% RSLogix 500 project Adaptive Fault-Resilient Robotic Pick-and-Place Cell.RSS, saved by version 8.30.00.16 %
PROJECT "UNTITLED"    % processor: Bul.1763 MicroLogix 1100 Series B %

PROGRAM FILES
  LAD 2 "MAIN/ARM"  15 rungs
  LAD 3 "SAFETY"  28 rungs
  LAD 4 "MODES"  4 rungs
  LAD 5 "DIGITAL IO"  17 rungs
  LAD 6 "ANALOG IO"  2 rungs
  LAD 7 "STATE"  6 rungs
  LAD 8 "SENSORS"  5 rungs
  LAD 9 "SYSTEM H"  6 rungs
  LAD 10 "H SAFETY"  6 rungs
  LAD 11 "H IO"  3 rungs
  LAD 12 "H STATE"  4 rungs
  LAD 13 "LOGIC"  19 rungs

DATA FILES
  O0 OUTPUT  7 elements
  I1 INPUT  14 elements
  S2 STATUS  66 elements
  B3 BINARY  10 elements
  T4 TIMER  8 elements
  C5 COUNTER  10 elements
  R6 CONTROL  1 elements
  N7 INTEGER  1 elements
  F8 FLOAT  1 elements

LADDER 2 "MAIN/ARM"
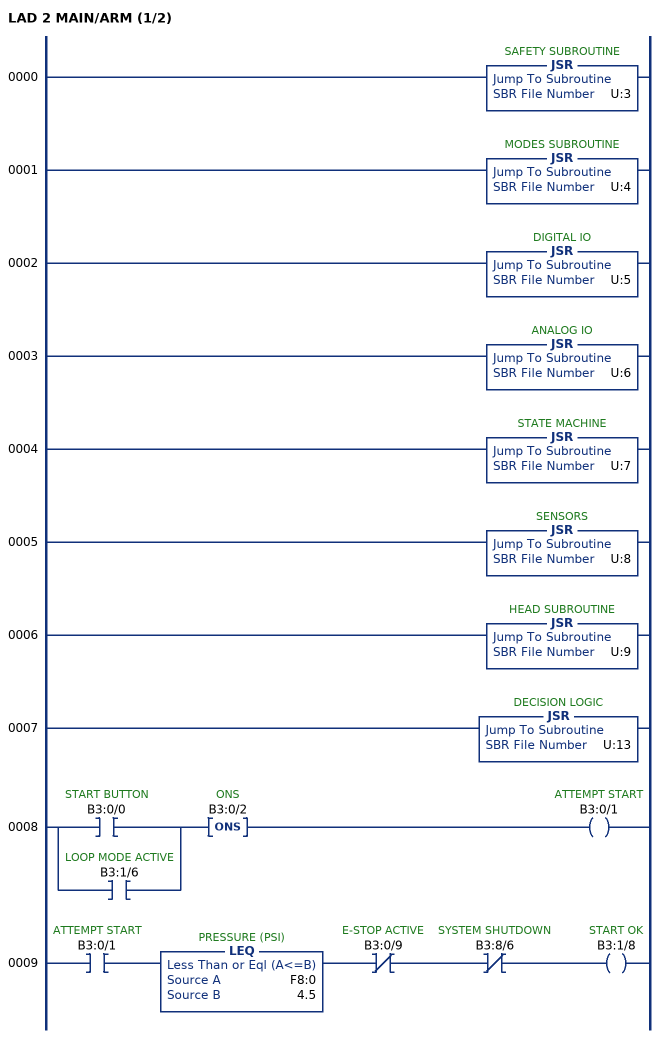
% Rung: 0 %
SOR JSR U:3 EOR
%   U:3  "SAFETY SUBROUTINE" %
% Rung: 1 %
SOR JSR U:4 EOR
%   U:4  "MODES SUBROUTINE" %
% Rung: 2 %
SOR JSR U:5 EOR
%   U:5  "DIGITAL IO" %
% Rung: 3 %
SOR JSR U:6 EOR
%   U:6  "ANALOG IO" %
% Rung: 4 %
SOR JSR U:7 EOR
%   U:7  "STATE MACHINE" %
% Rung: 5 %
SOR JSR U:8 EOR
%   U:8  "SENSORS" %
% Rung: 6 %
SOR JSR U:9 EOR
%   U:9  "HEAD SUBROUTINE" %
% Rung: 7 %
SOR JSR U:13 EOR
%   U:13  "DECISION LOGIC" %
% Rung: 8 %
SOR BST XIC B3:0/0 NXB XIC B3:1/6 BND ONS B3:0/2 OTE B3:0/1 EOR
%   B3:0/0  "START BUTTON" %
%   B3:1/6  "LOOP MODE ACTIVE" %
%   B3:0/2  "ONS" %
%   B3:0/1  "ATTEMPT START" %
% Rung: 9 %
SOR XIC B3:0/1 LEQ F8:0 4.5 XIO B3:0/9 XIO B3:8/6 OTE B3:1/8 EOR
%   B3:0/1  "ATTEMPT START" %
%   F8:0  "PRESSURE (PSI)" %
%   B3:0/9  "E-STOP ACTIVE" %
%   B3:8/6  "SYSTEM SHUTDOWN" %
%   B3:1/8  "START OK" %

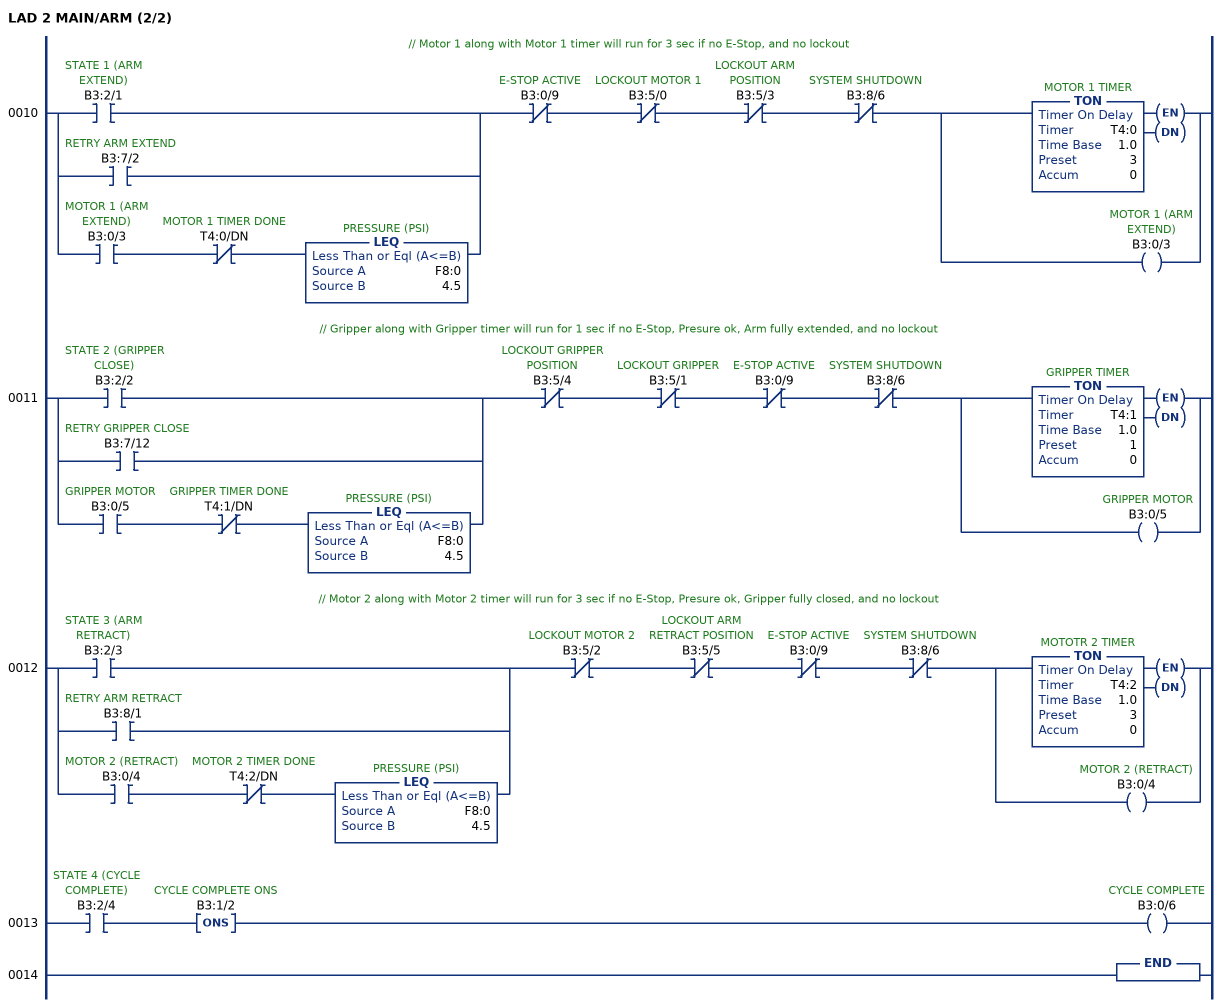
% Rung: 10 %
% // Motor 1 along with Motor 1 timer will run for 3 sec if no E-Stop, and no lockout %
SOR BST BST XIC B3:2/1 NXB XIC B3:7/2 BND NXB XIC B3:0/3 XIO T4:0/DN LEQ F8:0 4.5 BND XIO B3:0/9 XIO B3:5/0 XIO B3:5/3 XIO B3:8/6 BST TON T4:0 1.0 3 0 NXB OTE B3:0/3 BND EOR
%   B3:2/1  "STATE 1 (ARM EXTEND)" %
%   B3:7/2  "RETRY ARM EXTEND" %
%   B3:0/3  "MOTOR 1 (ARM EXTEND)" %
%   T4:0/DN  "MOTOR 1 TIMER DONE" %
%   F8:0  "PRESSURE (PSI)" %
%   B3:0/9  "E-STOP ACTIVE" %
%   B3:5/0  "LOCKOUT MOTOR 1" %
%   B3:5/3  "LOCKOUT ARM POSITION" %
%   B3:8/6  "SYSTEM SHUTDOWN" %
%   T4:0  "MOTOR 1 TIMER" %
% Rung: 11 %
% // Gripper along with Gripper timer will run for 1 sec if no E-Stop, Presure ok, Arm fully extended, and no lockout %
SOR BST BST XIC B3:2/2 NXB XIC B3:7/12 BND NXB XIC B3:0/5 XIO T4:1/DN LEQ F8:0 4.5 BND XIO B3:5/4 XIO B3:5/1 XIO B3:0/9 XIO B3:8/6 BST TON T4:1 1.0 1 0 NXB OTE B3:0/5 BND EOR
%   B3:2/2  "STATE 2 (GRIPPER CLOSE)" %
%   B3:7/12  "RETRY GRIPPER CLOSE" %
%   B3:0/5  "GRIPPER MOTOR" %
%   T4:1/DN  "GRIPPER TIMER DONE" %
%   F8:0  "PRESSURE (PSI)" %
%   B3:5/4  "LOCKOUT GRIPPER POSITION" %
%   B3:5/1  "LOCKOUT GRIPPER" %
%   B3:0/9  "E-STOP ACTIVE" %
%   B3:8/6  "SYSTEM SHUTDOWN" %
%   T4:1  "GRIPPER TIMER" %
% Rung: 12 %
% // Motor 2 along with Motor 2 timer will run for 3 sec if no E-Stop, Presure ok, Gripper fully closed, and no lockout %
SOR BST BST XIC B3:2/3 NXB XIC B3:8/1 BND NXB XIC B3:0/4 XIO T4:2/DN LEQ F8:0 4.5 BND XIO B3:5/2 XIO B3:5/5 XIO B3:0/9 XIO B3:8/6 BST TON T4:2 1.0 3 0 NXB OTE B3:0/4 BND EOR
%   B3:2/3  "STATE 3 (ARM RETRACT)" %
%   B3:8/1  "RETRY ARM RETRACT" %
%   B3:0/4  "MOTOR 2 (RETRACT)" %
%   T4:2/DN  "MOTOR 2 TIMER DONE" %
%   F8:0  "PRESSURE (PSI)" %
%   B3:5/2  "LOCKOUT MOTOR 2" %
%   B3:5/5  "LOCKOUT ARM RETRACT POSITION" %
%   B3:0/9  "E-STOP ACTIVE" %
%   B3:8/6  "SYSTEM SHUTDOWN" %
%   T4:2  "MOTOTR 2 TIMER" %
% Rung: 13 %
SOR XIC B3:2/4 ONS B3:1/2 OTE B3:0/6 EOR
%   B3:2/4  "STATE 4 (CYCLE COMPLETE)" %
%   B3:1/2  "CYCLE COMPLETE ONS" %
%   B3:0/6  "CYCLE COMPLETE" %
% Rung: 14 %
SOR END EOR

LADDER 3 "SAFETY"
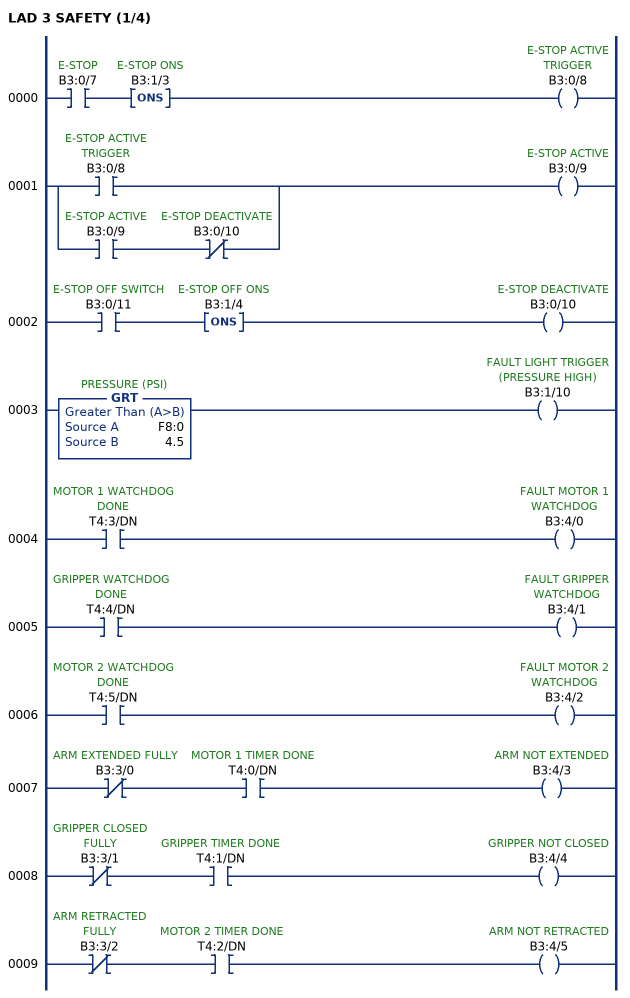
% Rung: 0 %
SOR XIC B3:0/7 ONS B3:1/3 OTE B3:0/8 EOR
%   B3:0/7  "E-STOP" %
%   B3:1/3  "E-STOP ONS" %
%   B3:0/8  "E-STOP ACTIVE TRIGGER" %
% Rung: 1 %
SOR BST XIC B3:0/8 NXB XIC B3:0/9 XIO B3:0/10 BND OTE B3:0/9 EOR
%   B3:0/8  "E-STOP ACTIVE TRIGGER" %
%   B3:0/9  "E-STOP ACTIVE" %
%   B3:0/10  "E-STOP DEACTIVATE" %
% Rung: 2 %
SOR XIC B3:0/11 ONS B3:1/4 OTE B3:0/10 EOR
%   B3:0/11  "E-STOP OFF SWITCH" %
%   B3:1/4  "E-STOP OFF ONS" %
%   B3:0/10  "E-STOP DEACTIVATE" %
% Rung: 3 %
SOR GRT F8:0 4.5 OTE B3:1/10 EOR
%   F8:0  "PRESSURE (PSI)" %
%   B3:1/10  "FAULT LIGHT TRIGGER (PRESSURE HIGH)" %
% Rung: 4 %
SOR XIC T4:3/DN OTE B3:4/0 EOR
%   T4:3/DN  "MOTOR 1 WATCHDOG DONE" %
%   B3:4/0  "FAULT MOTOR 1 WATCHDOG" %
% Rung: 5 %
SOR XIC T4:4/DN OTE B3:4/1 EOR
%   T4:4/DN  "GRIPPER WATCHDOG DONE" %
%   B3:4/1  "FAULT GRIPPER WATCHDOG" %
% Rung: 6 %
SOR XIC T4:5/DN OTE B3:4/2 EOR
%   T4:5/DN  "MOTOR 2 WATCHDOG DONE" %
%   B3:4/2  "FAULT MOTOR 2 WATCHDOG" %
% Rung: 7 %
SOR XIO B3:3/0 XIC T4:0/DN OTE B3:4/3 EOR
%   B3:3/0  "ARM EXTENDED FULLY" %
%   T4:0/DN  "MOTOR 1 TIMER DONE" %
%   B3:4/3  "ARM NOT EXTENDED" %
% Rung: 8 %
SOR XIO B3:3/1 XIC T4:1/DN OTE B3:4/4 EOR
%   B3:3/1  "GRIPPER CLOSED FULLY" %
%   T4:1/DN  "GRIPPER TIMER DONE" %
%   B3:4/4  "GRIPPER NOT CLOSED" %
% Rung: 9 %
SOR XIO B3:3/2 XIC T4:2/DN OTE B3:4/5 EOR
%   B3:3/2  "ARM RETRACTED FULLY" %
%   T4:2/DN  "MOTOR 2 TIMER DONE" %
%   B3:4/5  "ARM NOT RETRACTED" %

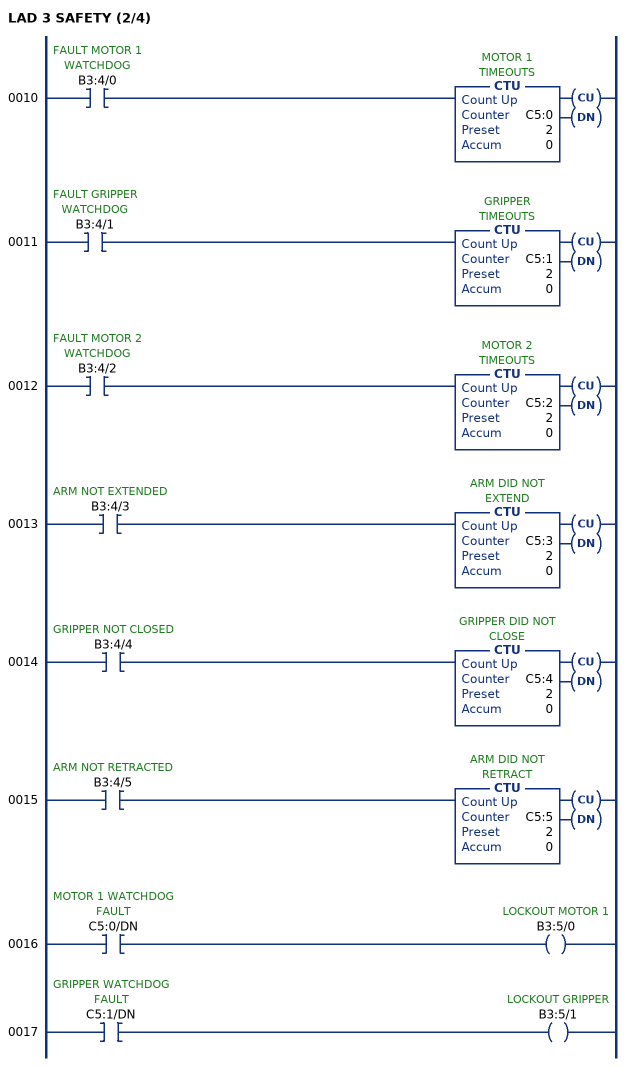
% Rung: 10 %
SOR XIC B3:4/0 CTU C5:0 2 0 EOR
%   B3:4/0  "FAULT MOTOR 1 WATCHDOG" %
%   C5:0  "MOTOR 1 TIMEOUTS" %
% Rung: 11 %
SOR XIC B3:4/1 CTU C5:1 2 0 EOR
%   B3:4/1  "FAULT GRIPPER WATCHDOG" %
%   C5:1  "GRIPPER TIMEOUTS" %
% Rung: 12 %
SOR XIC B3:4/2 CTU C5:2 2 0 EOR
%   B3:4/2  "FAULT MOTOR 2 WATCHDOG" %
%   C5:2  "MOTOR 2 TIMEOUTS" %
% Rung: 13 %
SOR XIC B3:4/3 CTU C5:3 2 0 EOR
%   B3:4/3  "ARM NOT EXTENDED" %
%   C5:3  "ARM DID NOT EXTEND" %
% Rung: 14 %
SOR XIC B3:4/4 CTU C5:4 2 0 EOR
%   B3:4/4  "GRIPPER NOT CLOSED" %
%   C5:4  "GRIPPER DID NOT CLOSE" %
% Rung: 15 %
SOR XIC B3:4/5 CTU C5:5 2 0 EOR
%   B3:4/5  "ARM NOT RETRACTED" %
%   C5:5  "ARM DID NOT RETRACT" %
% Rung: 16 %
SOR XIC C5:0/DN OTE B3:5/0 EOR
%   C5:0/DN  "MOTOR 1 WATCHDOG FAULT" %
%   B3:5/0  "LOCKOUT MOTOR 1" %
% Rung: 17 %
SOR XIC C5:1/DN OTE B3:5/1 EOR
%   C5:1/DN  "GRIPPER WATCHDOG FAULT" %
%   B3:5/1  "LOCKOUT GRIPPER" %

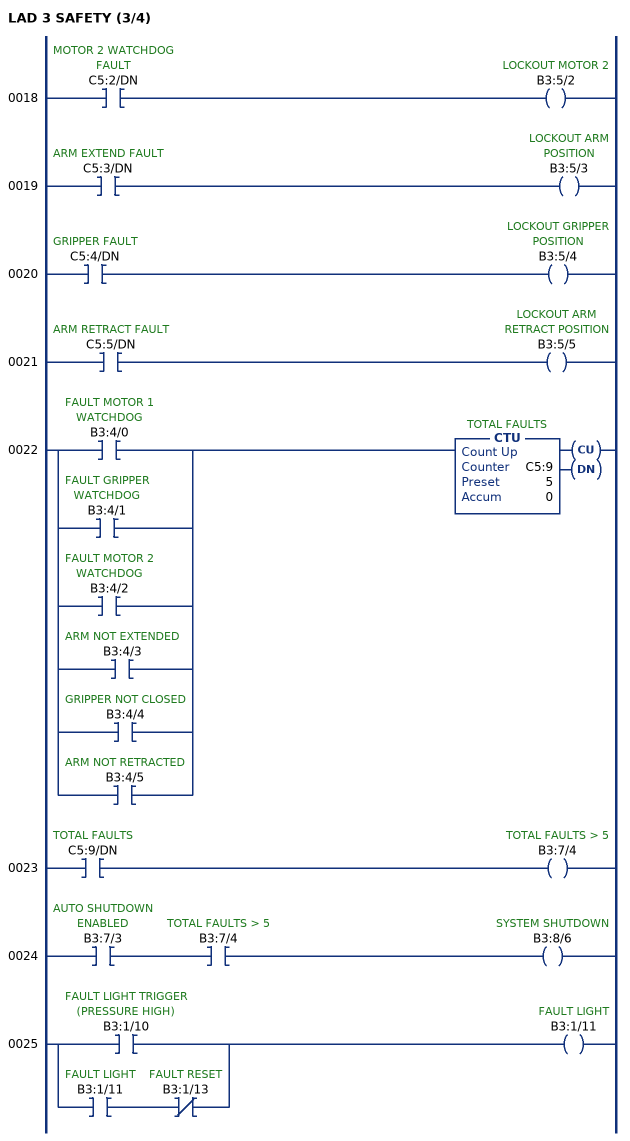
% Rung: 18 %
SOR XIC C5:2/DN OTE B3:5/2 EOR
%   C5:2/DN  "MOTOR 2 WATCHDOG FAULT" %
%   B3:5/2  "LOCKOUT MOTOR 2" %
% Rung: 19 %
SOR XIC C5:3/DN OTE B3:5/3 EOR
%   C5:3/DN  "ARM EXTEND FAULT" %
%   B3:5/3  "LOCKOUT ARM POSITION" %
% Rung: 20 %
SOR XIC C5:4/DN OTE B3:5/4 EOR
%   C5:4/DN  "GRIPPER FAULT" %
%   B3:5/4  "LOCKOUT GRIPPER POSITION" %
% Rung: 21 %
SOR XIC C5:5/DN OTE B3:5/5 EOR
%   C5:5/DN  "ARM RETRACT FAULT" %
%   B3:5/5  "LOCKOUT ARM RETRACT POSITION" %
% Rung: 22 %
SOR BST XIC B3:4/0 NXB XIC B3:4/1 NXB XIC B3:4/2 NXB XIC B3:4/3 NXB XIC B3:4/4 NXB XIC B3:4/5 BND CTU C5:9 5 0 EOR
%   B3:4/0  "FAULT MOTOR 1 WATCHDOG" %
%   B3:4/1  "FAULT GRIPPER WATCHDOG" %
%   B3:4/2  "FAULT MOTOR 2 WATCHDOG" %
%   B3:4/3  "ARM NOT EXTENDED" %
%   B3:4/4  "GRIPPER NOT CLOSED" %
%   B3:4/5  "ARM NOT RETRACTED" %
%   C5:9  "TOTAL FAULTS" %
% Rung: 23 %
SOR XIC C5:9/DN OTE B3:7/4 EOR
%   C5:9  "TOTAL FAULTS" %
%   B3:7/4  "TOTAL FAULTS > 5" %
% Rung: 24 %
SOR XIC B3:7/3 XIC B3:7/4 OTE B3:8/6 EOR
%   B3:7/3  "AUTO SHUTDOWN ENABLED" %
%   B3:7/4  "TOTAL FAULTS > 5" %
%   B3:8/6  "SYSTEM SHUTDOWN" %
% Rung: 25 %
SOR BST XIC B3:1/10 NXB XIC B3:1/11 XIO B3:1/13 BND OTE B3:1/11 EOR
%   B3:1/10  "FAULT LIGHT TRIGGER (PRESSURE HIGH)" %
%   B3:1/11  "FAULT LIGHT" %
%   B3:1/13  "FAULT RESET" %

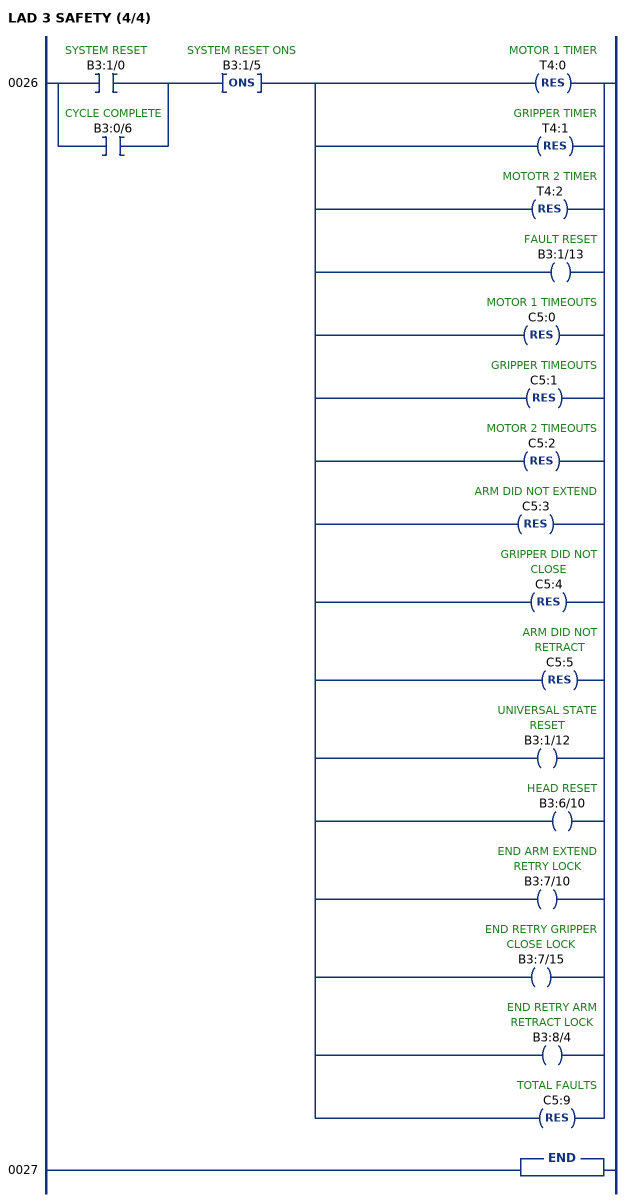
% Rung: 26 %
SOR BST XIC B3:1/0 NXB XIC B3:0/6 BND ONS B3:1/5 BST RES T4:0 NXB RES T4:1 NXB RES T4:2 NXB OTE B3:1/13 NXB RES C5:0 NXB RES C5:1 NXB RES C5:2 NXB RES C5:3 NXB RES C5:4 NXB RES C5:5 NXB OTE B3:1/12 NXB OTE B3:6/10 NXB OTE B3:7/10 NXB OTE B3:7/15 NXB OTE B3:8/4 NXB RES C5:9 BND EOR
%   B3:1/0  "SYSTEM RESET" %
%   B3:0/6  "CYCLE COMPLETE" %
%   B3:1/5  "SYSTEM RESET ONS" %
%   T4:0  "MOTOR 1 TIMER" %
%   T4:1  "GRIPPER TIMER" %
%   T4:2  "MOTOTR 2 TIMER" %
%   B3:1/13  "FAULT RESET" %
%   C5:0  "MOTOR 1 TIMEOUTS" %
%   C5:1  "GRIPPER TIMEOUTS" %
%   C5:2  "MOTOR 2 TIMEOUTS" %
%   C5:3  "ARM DID NOT EXTEND" %
%   C5:4  "GRIPPER DID NOT CLOSE" %
%   C5:5  "ARM DID NOT RETRACT" %
%   B3:1/12  "UNIVERSAL STATE RESET" %
%   B3:6/10  "HEAD RESET" %
%   B3:7/10  "END ARM EXTEND RETRY LOCK" %
%   B3:7/15  "END RETRY GRIPPER CLOSE LOCK" %
%   B3:8/4  "END RETRY ARM RETRACT LOCK" %
%   C5:9  "TOTAL FAULTS" %
% Rung: 27 %
SOR END EOR

LADDER 4 "MODES"
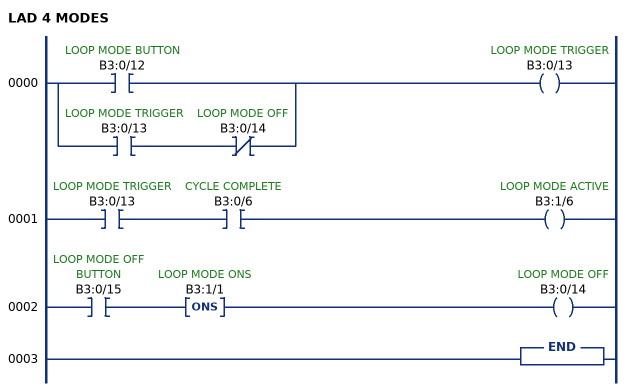
% Rung: 0 %
SOR BST XIC B3:0/12 NXB XIC B3:0/13 XIO B3:0/14 BND OTE B3:0/13 EOR
%   B3:0/12  "LOOP MODE BUTTON" %
%   B3:0/13  "LOOP MODE TRIGGER" %
%   B3:0/14  "LOOP MODE OFF" %
% Rung: 1 %
SOR XIC B3:0/13 XIC B3:0/6 OTE B3:1/6 EOR
%   B3:0/13  "LOOP MODE TRIGGER" %
%   B3:0/6  "CYCLE COMPLETE" %
%   B3:1/6  "LOOP MODE ACTIVE" %
% Rung: 2 %
SOR XIC B3:0/15 ONS B3:1/1 OTE B3:0/14 EOR
%   B3:0/15  "LOOP MODE OFF BUTTON" %
%   B3:1/1  "LOOP MODE ONS" %
%   B3:0/14  "LOOP MODE OFF" %
% Rung: 3 %
SOR END EOR

LADDER 5 "DIGITAL IO"
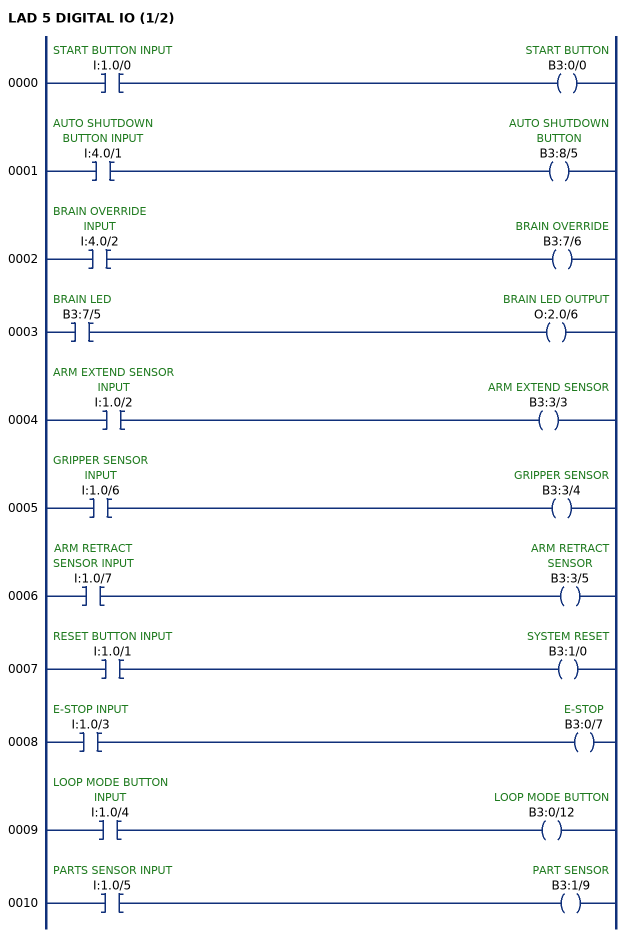
% Rung: 0 %
SOR XIC I:1.0/0 OTE B3:0/0 EOR
%   I:1.0/0  "START BUTTON INPUT" %
%   B3:0/0  "START BUTTON" %
% Rung: 1 %
SOR XIC I:4.0/1 OTE B3:8/5 EOR
%   I:4.0/1  "AUTO SHUTDOWN BUTTON INPUT" %
%   B3:8/5  "AUTO SHUTDOWN BUTTON" %
% Rung: 2 %
SOR XIC I:4.0/2 OTE B3:7/6 EOR
%   I:4.0/2  "BRAIN OVERRIDE INPUT" %
%   B3:7/6  "BRAIN OVERRIDE" %
% Rung: 3 %
SOR XIC B3:7/5 OTE O:2.0/6 EOR
%   B3:7/5  "BRAIN LED" %
%   O:2.0/6  "BRAIN LED OUTPUT" %
% Rung: 4 %
SOR XIC I:1.0/2 OTE B3:3/3 EOR
%   I:1.0/2  "ARM EXTEND SENSOR INPUT" %
%   B3:3/3  "ARM EXTEND SENSOR" %
% Rung: 5 %
SOR XIC I:1.0/6 OTE B3:3/4 EOR
%   I:1.0/6  "GRIPPER SENSOR INPUT" %
%   B3:3/4  "GRIPPER SENSOR" %
% Rung: 6 %
SOR XIC I:1.0/7 OTE B3:3/5 EOR
%   I:1.0/7  "ARM RETRACT SENSOR INPUT" %
%   B3:3/5  "ARM RETRACT SENSOR" %
% Rung: 7 %
SOR XIC I:1.0/1 OTE B3:1/0 EOR
%   I:1.0/1  "RESET BUTTON INPUT" %
%   B3:1/0  "SYSTEM RESET" %
% Rung: 8 %
SOR XIC I:1.0/3 OTE B3:0/7 EOR
%   I:1.0/3  "E-STOP INPUT" %
%   B3:0/7  "E-STOP" %
% Rung: 9 %
SOR XIC I:1.0/4 OTE B3:0/12 EOR
%   I:1.0/4  "LOOP MODE BUTTON INPUT" %
%   B3:0/12  "LOOP MODE BUTTON" %
% Rung: 10 %
SOR XIC I:1.0/5 OTE B3:1/9 EOR
%   I:1.0/5  "PARTS SENSOR INPUT" %
%   B3:1/9  "PART SENSOR" %

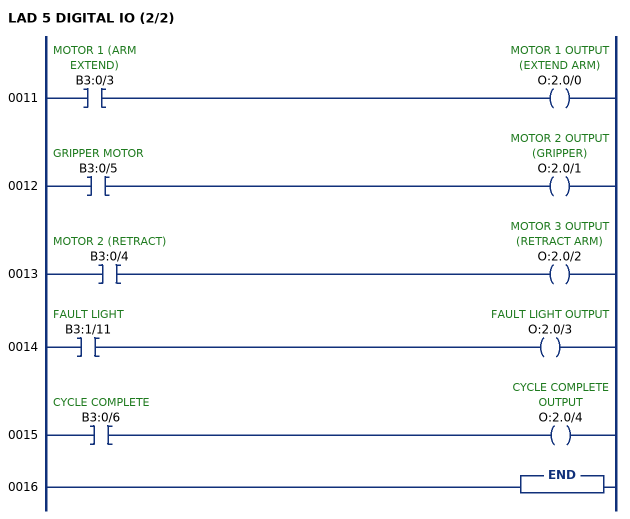
% Rung: 11 %
SOR XIC B3:0/3 OTE O:2.0/0 EOR
%   B3:0/3  "MOTOR 1 (ARM EXTEND)" %
%   O:2.0/0  "MOTOR 1 OUTPUT (EXTEND ARM)" %
% Rung: 12 %
SOR XIC B3:0/5 OTE O:2.0/1 EOR
%   B3:0/5  "GRIPPER MOTOR" %
%   O:2.0/1  "MOTOR 2 OUTPUT (GRIPPER)" %
% Rung: 13 %
SOR XIC B3:0/4 OTE O:2.0/2 EOR
%   B3:0/4  "MOTOR 2 (RETRACT)" %
%   O:2.0/2  "MOTOR 3 OUTPUT (RETRACT ARM)" %
% Rung: 14 %
SOR XIC B3:1/11 OTE O:2.0/3 EOR
%   B3:1/11  "FAULT LIGHT" %
%   O:2.0/3  "FAULT LIGHT OUTPUT" %
% Rung: 15 %
SOR XIC B3:0/6 OTE O:2.0/4 EOR
%   B3:0/6  "CYCLE COMPLETE" %
%   O:2.0/4  "CYCLE COMPLETE OUTPUT" %
% Rung: 16 %
SOR END EOR

LADDER 6 "ANALOG IO"
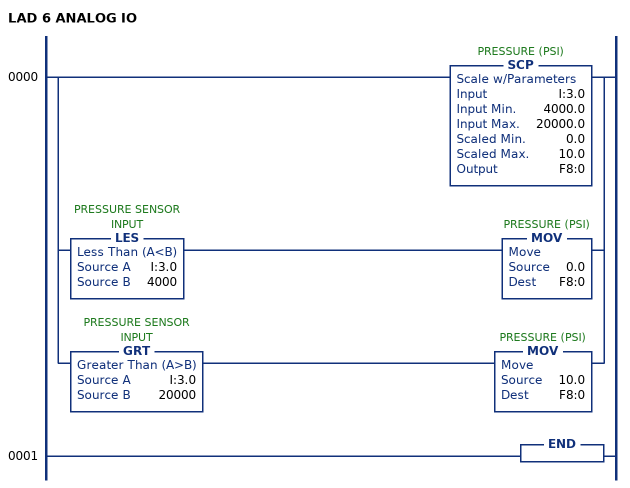
% Rung: 0 %
SOR BST SCP I:3.0 4000.0 20000.0 0.0 10.0 F8:0 NXB LES I:3.0 4000 MOV 0.0 F8:0 NXB GRT I:3.0 20000 MOV 10.0 F8:0 BND EOR
%   I:3.0  "PRESSURE SENSOR INPUT" %
%   F8:0  "PRESSURE (PSI)" %
% Rung: 1 %
SOR END EOR

LADDER 7 "STATE"
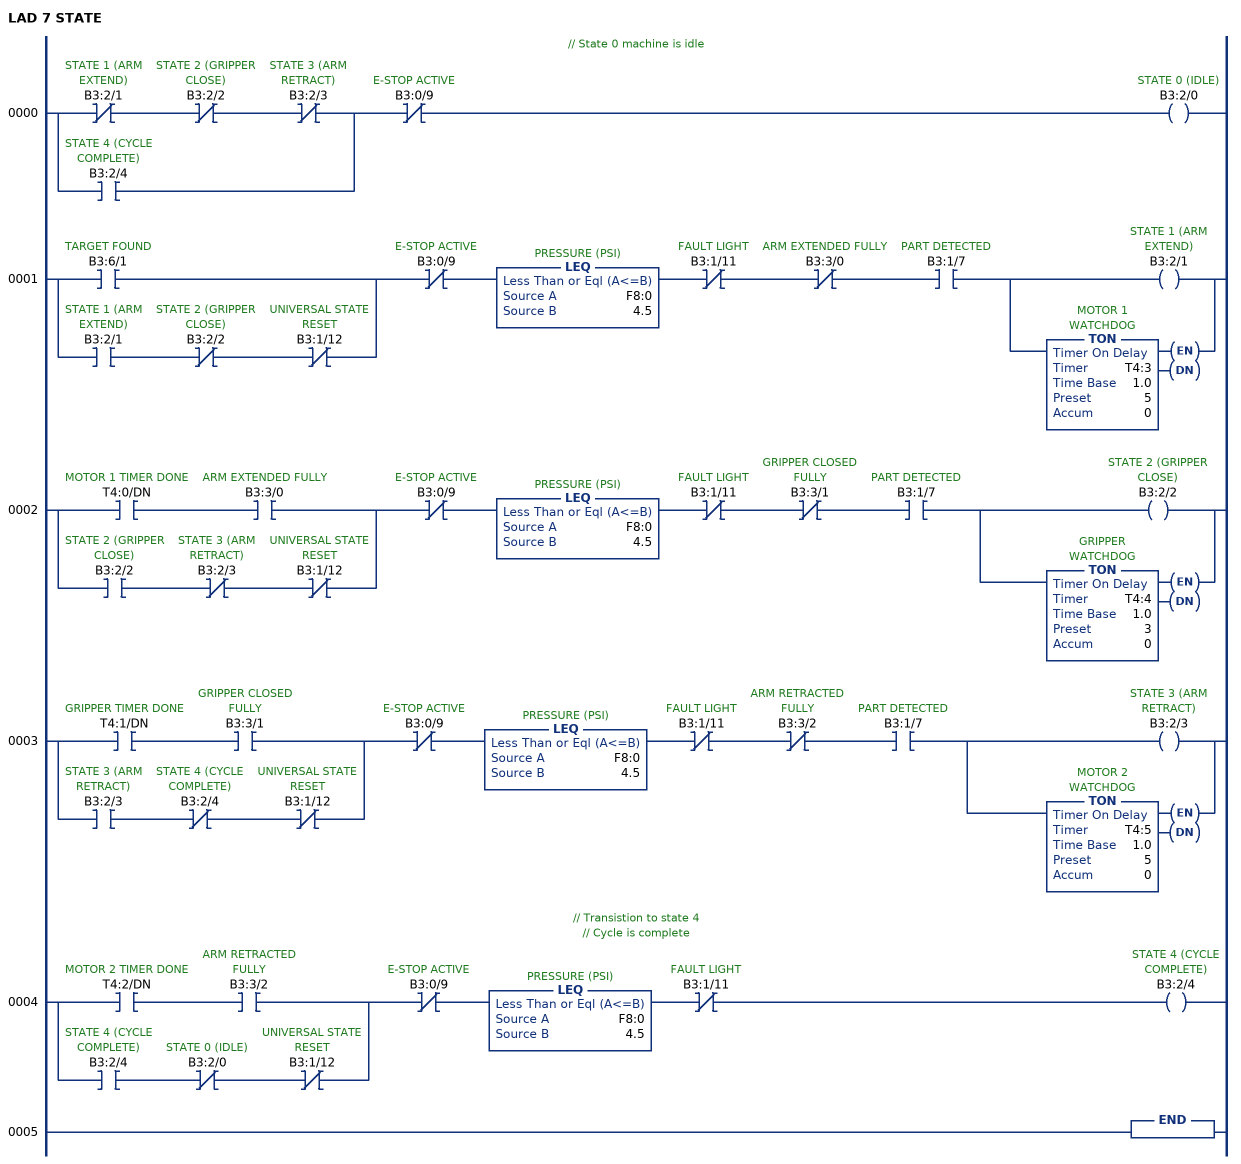
% Rung: 0 %
% // State 0 machine is idle %
SOR BST XIO B3:2/1 XIO B3:2/2 XIO B3:2/3 NXB XIC B3:2/4 BND XIO B3:0/9 OTE B3:2/0 EOR
%   B3:2/1  "STATE 1 (ARM EXTEND)" %
%   B3:2/2  "STATE 2 (GRIPPER CLOSE)" %
%   B3:2/3  "STATE 3 (ARM RETRACT)" %
%   B3:2/4  "STATE 4 (CYCLE COMPLETE)" %
%   B3:0/9  "E-STOP ACTIVE" %
%   B3:2/0  "STATE 0 (IDLE)" %
% Rung: 1 %
SOR BST XIC B3:6/1 NXB XIC B3:2/1 XIO B3:2/2 XIO B3:1/12 BND XIO B3:0/9 LEQ F8:0 4.5 XIO B3:1/11 XIO B3:3/0 XIC B3:1/7 BST OTE B3:2/1 NXB TON T4:3 1.0 5 0 BND EOR
%   B3:6/1  "TARGET FOUND" %
%   B3:2/1  "STATE 1 (ARM EXTEND)" %
%   B3:2/2  "STATE 2 (GRIPPER CLOSE)" %
%   B3:1/12  "UNIVERSAL STATE RESET" %
%   B3:0/9  "E-STOP ACTIVE" %
%   F8:0  "PRESSURE (PSI)" %
%   B3:1/11  "FAULT LIGHT" %
%   B3:3/0  "ARM EXTENDED FULLY" %
%   B3:1/7  "PART DETECTED" %
%   T4:3  "MOTOR 1 WATCHDOG" %
% Rung: 2 %
SOR BST XIC T4:0/DN XIC B3:3/0 NXB XIC B3:2/2 XIO B3:2/3 XIO B3:1/12 BND XIO B3:0/9 LEQ F8:0 4.5 XIO B3:1/11 XIO B3:3/1 XIC B3:1/7 BST OTE B3:2/2 NXB TON T4:4 1.0 3 0 BND EOR
%   T4:0/DN  "MOTOR 1 TIMER DONE" %
%   B3:3/0  "ARM EXTENDED FULLY" %
%   B3:2/2  "STATE 2 (GRIPPER CLOSE)" %
%   B3:2/3  "STATE 3 (ARM RETRACT)" %
%   B3:1/12  "UNIVERSAL STATE RESET" %
%   B3:0/9  "E-STOP ACTIVE" %
%   F8:0  "PRESSURE (PSI)" %
%   B3:1/11  "FAULT LIGHT" %
%   B3:3/1  "GRIPPER CLOSED FULLY" %
%   B3:1/7  "PART DETECTED" %
%   T4:4  "GRIPPER WATCHDOG" %
% Rung: 3 %
SOR BST XIC T4:1/DN XIC B3:3/1 NXB XIC B3:2/3 XIO B3:2/4 XIO B3:1/12 BND XIO B3:0/9 LEQ F8:0 4.5 XIO B3:1/11 XIO B3:3/2 XIC B3:1/7 BST OTE B3:2/3 NXB TON T4:5 1.0 5 0 BND EOR
%   T4:1/DN  "GRIPPER TIMER DONE" %
%   B3:3/1  "GRIPPER CLOSED FULLY" %
%   B3:2/3  "STATE 3 (ARM RETRACT)" %
%   B3:2/4  "STATE 4 (CYCLE COMPLETE)" %
%   B3:1/12  "UNIVERSAL STATE RESET" %
%   B3:0/9  "E-STOP ACTIVE" %
%   F8:0  "PRESSURE (PSI)" %
%   B3:1/11  "FAULT LIGHT" %
%   B3:3/2  "ARM RETRACTED FULLY" %
%   B3:1/7  "PART DETECTED" %
%   T4:5  "MOTOR 2 WATCHDOG" %
% Rung: 4 %
% // Transistion to state 4
% // Cycle is complete %
SOR BST XIC T4:2/DN XIC B3:3/2 NXB XIC B3:2/4 XIO B3:2/0 XIO B3:1/12 BND XIO B3:0/9 LEQ F8:0 4.5 XIO B3:1/11 OTE B3:2/4 EOR
%   T4:2/DN  "MOTOR 2 TIMER DONE" %
%   B3:3/2  "ARM RETRACTED FULLY" %
%   B3:2/4  "STATE 4 (CYCLE COMPLETE)" %
%   B3:2/0  "STATE 0 (IDLE)" %
%   B3:1/12  "UNIVERSAL STATE RESET" %
%   B3:0/9  "E-STOP ACTIVE" %
%   F8:0  "PRESSURE (PSI)" %
%   B3:1/11  "FAULT LIGHT" %
% Rung: 5 %
SOR END EOR

LADDER 8 "SENSORS"
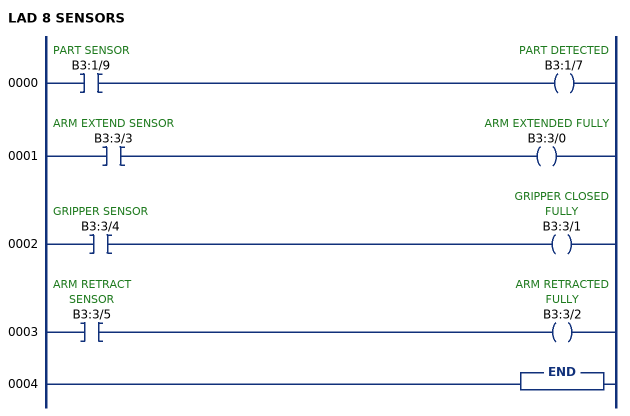
% Rung: 0 %
SOR XIC B3:1/9 OTE B3:1/7 EOR
%   B3:1/9  "PART SENSOR" %
%   B3:1/7  "PART DETECTED" %
% Rung: 1 %
SOR XIC B3:3/3 OTE B3:3/0 EOR
%   B3:3/3  "ARM EXTEND SENSOR" %
%   B3:3/0  "ARM EXTENDED FULLY" %
% Rung: 2 %
SOR XIC B3:3/4 OTE B3:3/1 EOR
%   B3:3/4  "GRIPPER SENSOR" %
%   B3:3/1  "GRIPPER CLOSED FULLY" %
% Rung: 3 %
SOR XIC B3:3/5 OTE B3:3/2 EOR
%   B3:3/5  "ARM RETRACT SENSOR" %
%   B3:3/2  "ARM RETRACTED FULLY" %
% Rung: 4 %
SOR END EOR

LADDER 9 "SYSTEM H"
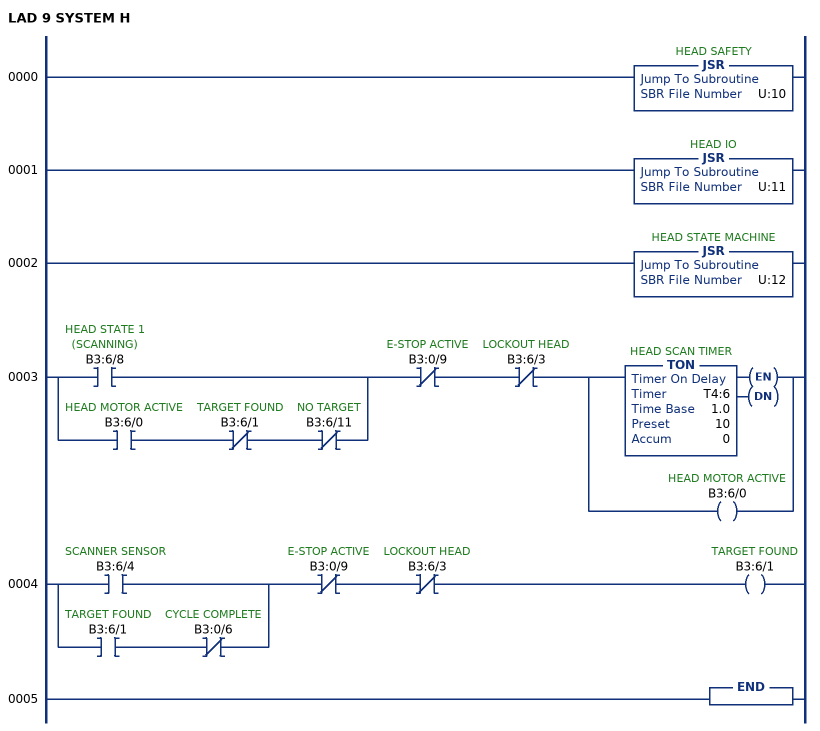
% Rung: 0 %
SOR JSR U:10 EOR
%   U:10  "HEAD SAFETY" %
% Rung: 1 %
SOR JSR U:11 EOR
%   U:11  "HEAD IO" %
% Rung: 2 %
SOR JSR U:12 EOR
%   U:12  "HEAD STATE MACHINE" %
% Rung: 3 %
SOR BST XIC B3:6/8 NXB XIC B3:6/0 XIO B3:6/1 XIO B3:6/11 BND XIO B3:0/9 XIO B3:6/3 BST TON T4:6 1.0 10 0 NXB OTE B3:6/0 BND EOR
%   B3:6/8  "HEAD STATE 1 (SCANNING)" %
%   B3:6/0  "HEAD MOTOR ACTIVE" %
%   B3:6/1  "TARGET FOUND" %
%   B3:6/11  "NO TARGET" %
%   B3:0/9  "E-STOP ACTIVE" %
%   B3:6/3  "LOCKOUT HEAD" %
%   T4:6  "HEAD SCAN TIMER" %
% Rung: 4 %
SOR BST XIC B3:6/4 NXB XIC B3:6/1 XIO B3:0/6 BND XIO B3:0/9 XIO B3:6/3 OTE B3:6/1 EOR
%   B3:6/4  "SCANNER SENSOR" %
%   B3:6/1  "TARGET FOUND" %
%   B3:0/6  "CYCLE COMPLETE" %
%   B3:0/9  "E-STOP ACTIVE" %
%   B3:6/3  "LOCKOUT HEAD" %
% Rung: 5 %
SOR END EOR

LADDER 10 "H SAFETY"
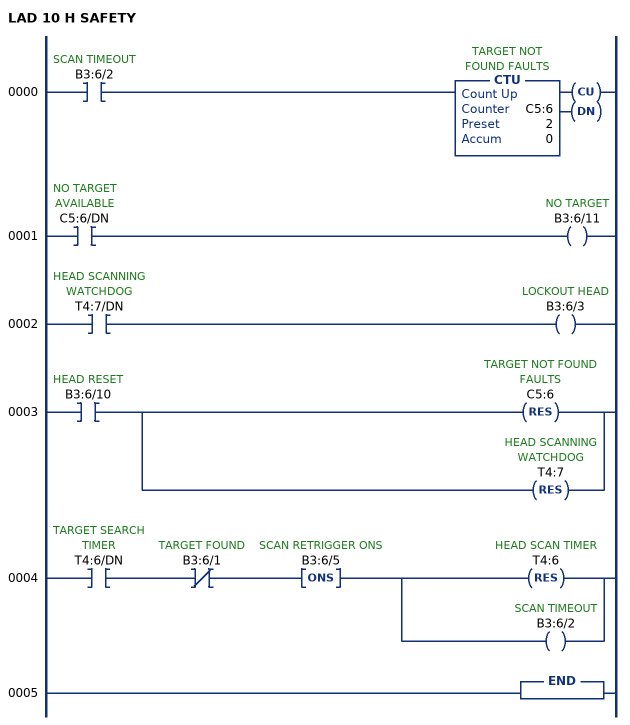
% Rung: 0 %
SOR XIC B3:6/2 CTU C5:6 2 0 EOR
%   B3:6/2  "SCAN TIMEOUT" %
%   C5:6  "TARGET NOT FOUND FAULTS" %
% Rung: 1 %
SOR XIC C5:6/DN OTE B3:6/11 EOR
%   C5:6/DN  "NO TARGET AVAILABLE" %
%   B3:6/11  "NO TARGET" %
% Rung: 2 %
SOR XIC T4:7/DN OTE B3:6/3 EOR
%   T4:7  "HEAD SCANNING WATCHDOG" %
%   B3:6/3  "LOCKOUT HEAD" %
% Rung: 3 %
SOR XIC B3:6/10 BST RES C5:6 NXB RES T4:7 BND EOR
%   B3:6/10  "HEAD RESET" %
%   C5:6  "TARGET NOT FOUND FAULTS" %
%   T4:7  "HEAD SCANNING WATCHDOG" %
% Rung: 4 %
SOR XIC T4:6/DN XIO B3:6/1 ONS B3:6/5 BST RES T4:6 NXB OTE B3:6/2 BND EOR
%   T4:6/DN  "TARGET SEARCH TIMER" %
%   B3:6/1  "TARGET FOUND" %
%   B3:6/5  "SCAN RETRIGGER ONS" %
%   T4:6  "HEAD SCAN TIMER" %
%   B3:6/2  "SCAN TIMEOUT" %
% Rung: 5 %
SOR END EOR

LADDER 11 "H IO"
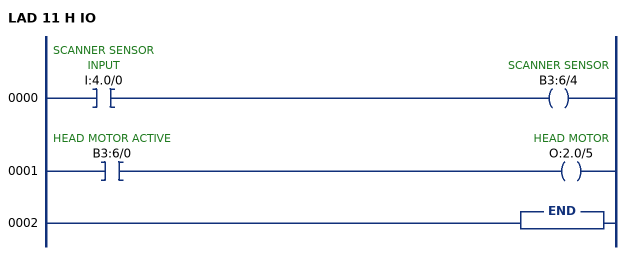
% Rung: 0 %
SOR XIC I:4.0/0 OTE B3:6/4 EOR
%   I:4.0/0  "SCANNER SENSOR INPUT" %
%   B3:6/4  "SCANNER SENSOR" %
% Rung: 1 %
SOR XIC B3:6/0 OTE O:2.0/5 EOR
%   B3:6/0  "HEAD MOTOR ACTIVE" %
%   O:2.0/5  "HEAD MOTOR" %
% Rung: 2 %
SOR END EOR

LADDER 12 "H STATE"
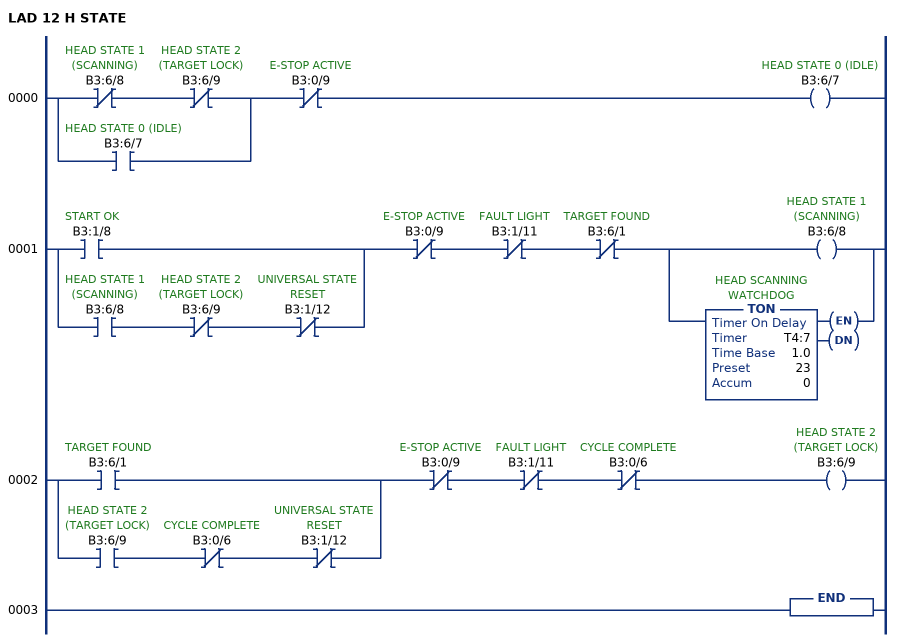
% Rung: 0 %
SOR BST XIO B3:6/8 XIO B3:6/9 NXB XIC B3:6/7 BND XIO B3:0/9 OTE B3:6/7 EOR
%   B3:6/8  "HEAD STATE 1 (SCANNING)" %
%   B3:6/9  "HEAD STATE 2 (TARGET LOCK)" %
%   B3:6/7  "HEAD STATE 0 (IDLE)" %
%   B3:0/9  "E-STOP ACTIVE" %
% Rung: 1 %
SOR BST XIC B3:1/8 NXB XIC B3:6/8 XIO B3:6/9 XIO B3:1/12 BND XIO B3:0/9 XIO B3:1/11 XIO B3:6/1 BST OTE B3:6/8 NXB TON T4:7 1.0 23 0 BND EOR
%   B3:1/8  "START OK" %
%   B3:6/8  "HEAD STATE 1 (SCANNING)" %
%   B3:6/9  "HEAD STATE 2 (TARGET LOCK)" %
%   B3:1/12  "UNIVERSAL STATE RESET" %
%   B3:0/9  "E-STOP ACTIVE" %
%   B3:1/11  "FAULT LIGHT" %
%   B3:6/1  "TARGET FOUND" %
%   T4:7  "HEAD SCANNING WATCHDOG" %
% Rung: 2 %
SOR BST XIC B3:6/1 NXB XIC B3:6/9 XIO B3:0/6 XIO B3:1/12 BND XIO B3:0/9 XIO B3:1/11 XIO B3:0/6 OTE B3:6/9 EOR
%   B3:6/1  "TARGET FOUND" %
%   B3:6/9  "HEAD STATE 2 (TARGET LOCK)" %
%   B3:0/6  "CYCLE COMPLETE" %
%   B3:1/12  "UNIVERSAL STATE RESET" %
%   B3:0/9  "E-STOP ACTIVE" %
%   B3:1/11  "FAULT LIGHT" %
% Rung: 3 %
SOR END EOR

LADDER 13 "LOGIC"
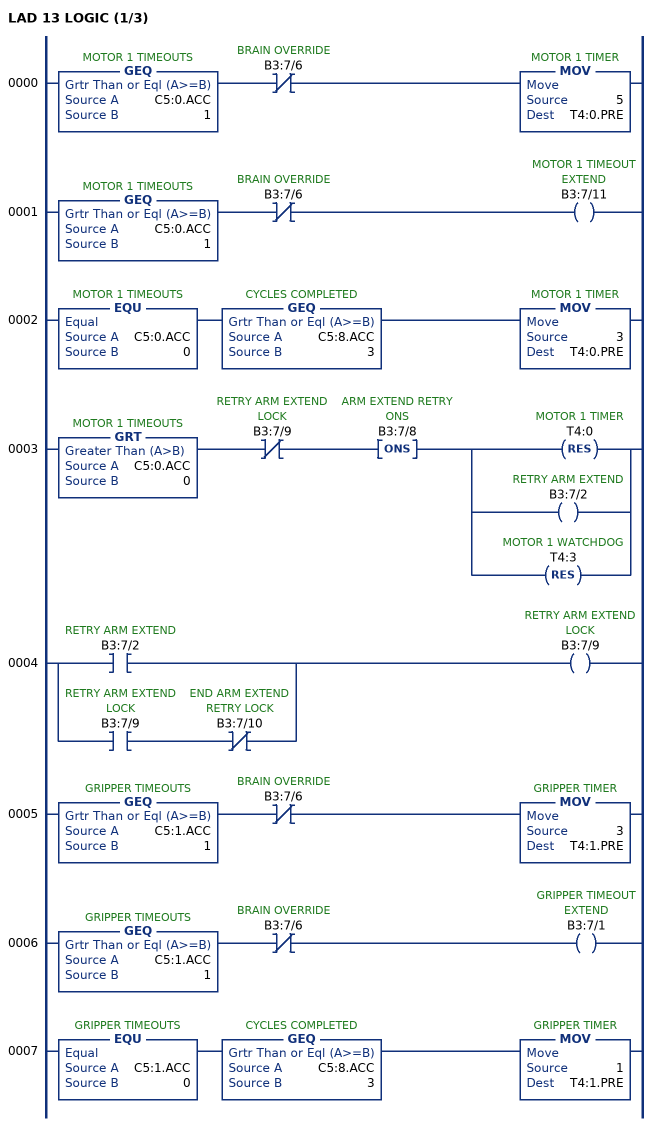
% Rung: 0 %
SOR GEQ C5:0.ACC 1 XIO B3:7/6 MOV 5 T4:0.PRE EOR
%   C5:0  "MOTOR 1 TIMEOUTS" %
%   B3:7/6  "BRAIN OVERRIDE" %
%   T4:0  "MOTOR 1 TIMER" %
% Rung: 1 %
SOR GEQ C5:0.ACC 1 XIO B3:7/6 OTE B3:7/11 EOR
%   C5:0  "MOTOR 1 TIMEOUTS" %
%   B3:7/6  "BRAIN OVERRIDE" %
%   B3:7/11  "MOTOR 1 TIMEOUT EXTEND" %
% Rung: 2 %
SOR EQU C5:0.ACC 0 GEQ C5:8.ACC 3 MOV 3 T4:0.PRE EOR
%   C5:0  "MOTOR 1 TIMEOUTS" %
%   C5:8.ACC  "CYCLES COMPLETED" %
%   T4:0  "MOTOR 1 TIMER" %
% Rung: 3 %
SOR GRT C5:0.ACC 0 XIO B3:7/9 ONS B3:7/8 BST RES T4:0 NXB OTE B3:7/2 NXB RES T4:3 BND EOR
%   C5:0  "MOTOR 1 TIMEOUTS" %
%   B3:7/9  "RETRY ARM EXTEND LOCK" %
%   B3:7/8  "ARM EXTEND RETRY ONS" %
%   T4:0  "MOTOR 1 TIMER" %
%   B3:7/2  "RETRY ARM EXTEND" %
%   T4:3  "MOTOR 1 WATCHDOG" %
% Rung: 4 %
SOR BST XIC B3:7/2 NXB XIC B3:7/9 XIO B3:7/10 BND OTE B3:7/9 EOR
%   B3:7/2  "RETRY ARM EXTEND" %
%   B3:7/9  "RETRY ARM EXTEND LOCK" %
%   B3:7/10  "END ARM EXTEND RETRY LOCK" %
% Rung: 5 %
SOR GEQ C5:1.ACC 1 XIO B3:7/6 MOV 3 T4:1.PRE EOR
%   C5:1  "GRIPPER TIMEOUTS" %
%   B3:7/6  "BRAIN OVERRIDE" %
%   T4:1  "GRIPPER TIMER" %
% Rung: 6 %
SOR GEQ C5:1.ACC 1 XIO B3:7/6 OTE B3:7/1 EOR
%   C5:1  "GRIPPER TIMEOUTS" %
%   B3:7/6  "BRAIN OVERRIDE" %
%   B3:7/1  "GRIPPER TIMEOUT EXTEND" %
% Rung: 7 %
SOR EQU C5:1.ACC 0 GEQ C5:8.ACC 3 MOV 1 T4:1.PRE EOR
%   C5:1  "GRIPPER TIMEOUTS" %
%   C5:8.ACC  "CYCLES COMPLETED" %
%   T4:1  "GRIPPER TIMER" %

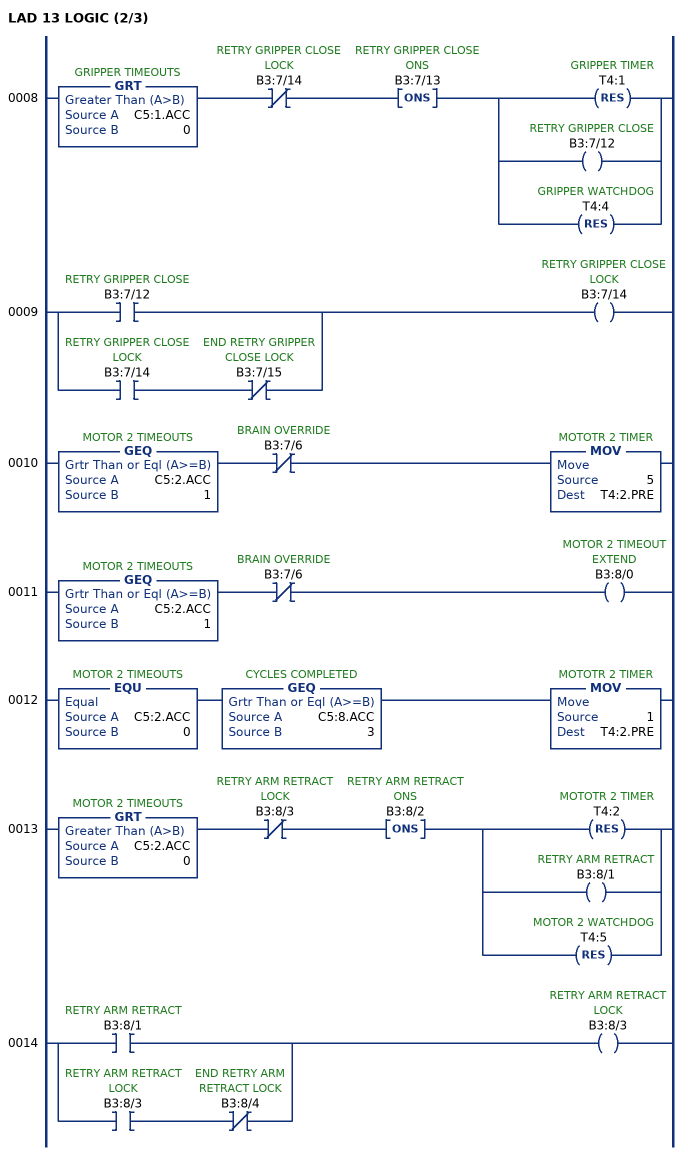
% Rung: 8 %
SOR GRT C5:1.ACC 0 XIO B3:7/14 ONS B3:7/13 BST RES T4:1 NXB OTE B3:7/12 NXB RES T4:4 BND EOR
%   C5:1  "GRIPPER TIMEOUTS" %
%   B3:7/14  "RETRY GRIPPER CLOSE LOCK" %
%   B3:7/13  "RETRY GRIPPER CLOSE ONS" %
%   T4:1  "GRIPPER TIMER" %
%   B3:7/12  "RETRY GRIPPER CLOSE" %
%   T4:4  "GRIPPER WATCHDOG" %
% Rung: 9 %
SOR BST XIC B3:7/12 NXB XIC B3:7/14 XIO B3:7/15 BND OTE B3:7/14 EOR
%   B3:7/12  "RETRY GRIPPER CLOSE" %
%   B3:7/14  "RETRY GRIPPER CLOSE LOCK" %
%   B3:7/15  "END RETRY GRIPPER CLOSE LOCK" %
% Rung: 10 %
SOR GEQ C5:2.ACC 1 XIO B3:7/6 MOV 5 T4:2.PRE EOR
%   C5:2  "MOTOR 2 TIMEOUTS" %
%   B3:7/6  "BRAIN OVERRIDE" %
%   T4:2  "MOTOTR 2 TIMER" %
% Rung: 11 %
SOR GEQ C5:2.ACC 1 XIO B3:7/6 OTE B3:8/0 EOR
%   C5:2  "MOTOR 2 TIMEOUTS" %
%   B3:7/6  "BRAIN OVERRIDE" %
%   B3:8/0  "MOTOR 2 TIMEOUT EXTEND" %
% Rung: 12 %
SOR EQU C5:2.ACC 0 GEQ C5:8.ACC 3 MOV 1 T4:2.PRE EOR
%   C5:2  "MOTOR 2 TIMEOUTS" %
%   C5:8.ACC  "CYCLES COMPLETED" %
%   T4:2  "MOTOTR 2 TIMER" %
% Rung: 13 %
SOR GRT C5:2.ACC 0 XIO B3:8/3 ONS B3:8/2 BST RES T4:2 NXB OTE B3:8/1 NXB RES T4:5 BND EOR
%   C5:2  "MOTOR 2 TIMEOUTS" %
%   B3:8/3  "RETRY ARM RETRACT LOCK" %
%   B3:8/2  "RETRY ARM RETRACT ONS" %
%   T4:2  "MOTOTR 2 TIMER" %
%   B3:8/1  "RETRY ARM RETRACT" %
%   T4:5  "MOTOR 2 WATCHDOG" %
% Rung: 14 %
SOR BST XIC B3:8/1 NXB XIC B3:8/3 XIO B3:8/4 BND OTE B3:8/3 EOR
%   B3:8/1  "RETRY ARM RETRACT" %
%   B3:8/3  "RETRY ARM RETRACT LOCK" %
%   B3:8/4  "END RETRY ARM RETRACT LOCK" %

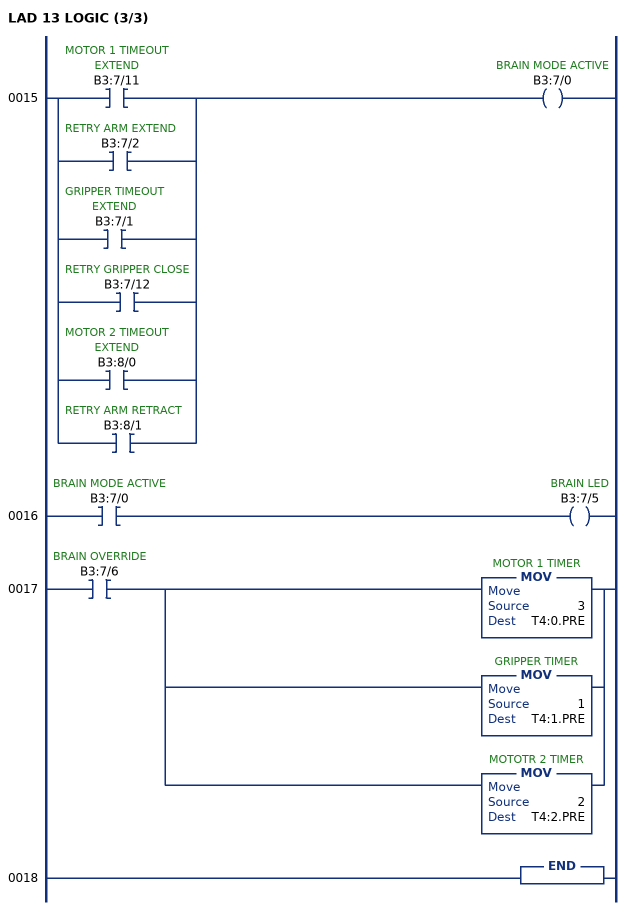
% Rung: 15 %
SOR BST XIC B3:7/11 NXB XIC B3:7/2 NXB XIC B3:7/1 NXB XIC B3:7/12 NXB XIC B3:8/0 NXB XIC B3:8/1 BND OTE B3:7/0 EOR
%   B3:7/11  "MOTOR 1 TIMEOUT EXTEND" %
%   B3:7/2  "RETRY ARM EXTEND" %
%   B3:7/1  "GRIPPER TIMEOUT EXTEND" %
%   B3:7/12  "RETRY GRIPPER CLOSE" %
%   B3:8/0  "MOTOR 2 TIMEOUT EXTEND" %
%   B3:8/1  "RETRY ARM RETRACT" %
%   B3:7/0  "BRAIN MODE ACTIVE" %
% Rung: 16 %
SOR XIC B3:7/0 OTE B3:7/5 EOR
%   B3:7/0  "BRAIN MODE ACTIVE" %
%   B3:7/5  "BRAIN LED" %
% Rung: 17 %
SOR XIC B3:7/6 BST MOV 3 T4:0.PRE NXB MOV 1 T4:1.PRE NXB MOV 2 T4:2.PRE BND EOR
%   B3:7/6  "BRAIN OVERRIDE" %
%   T4:0  "MOTOR 1 TIMER" %
%   T4:1  "GRIPPER TIMER" %
%   T4:2  "MOTOTR 2 TIMER" %
% Rung: 18 %
SOR END EOR

OTHER DOCUMENTED ADDRESSES
  B3:6/6  "SCAN ACTIVE"
  B3:7/7  "SYSTEM LOCK"
  C5:7  "SCANNER WATCHDOG TIME OUT"
  C5:8  "CYCLES COMPLETED COUNTER"
  C5:8/DN  "CYCLES COMPLETED MAX COUNT"
  I:3.0/0  "PRESSURE SENSOR INPUT"

COMMENTS NOT ATTACHED TO A CURRENT RUNG
  C5:8: //Track number of cycles completed to 100 then reset cycle complete counter

DATA TABLE (non-zero values as saved)
DATA T4
% .PRE .ACC %
% T4:0 % 3 0
% T4:1 % 1 0
% T4:2 % 3 0
% T4:3 % 5 0
% T4:4 % 3 0
% T4:5 % 5 0
% T4:6 % 10 0
% T4:7 % 23 0
DATA C5
% .PRE .ACC %
% C5:0 % 2 0
% C5:1 % 2 0
% C5:2 % 2 0
% C5:3 % 2 0
% C5:4 % 2 0
% C5:5 % 2 0
% C5:6 % 2 0
% C5:9 % 5 0
